(* PLC project Unnamed, Unknown Unnamed 1 *)
(* stored: creationDateTime 2026-03-27T23:35:05, modificationDateTime 2026-03-27T23:35:05 *)

PROGRAM main
  VAR
    start AT %IX0.0 : BOOL;
    stop AT %IX0.1 : BOOL;
    led AT %QX0.0 : BOOL;
  END_VAR
  VAR
    coil : BOOL;
    TON0 : TON;
    TOF0 : TOF;
  END_VAR

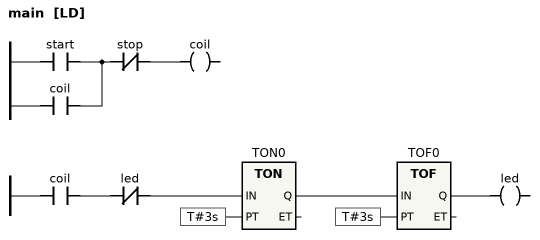
(* LD diagram, written out as Structured Text *)
coil := (start OR coil) AND NOT stop;
TON0(IN := coil AND NOT led, PT := T#3s);
TOF0(IN := TON0.Q, PT := T#3s);
led := TOF0.Q;
END_PROGRAM

CONFIGURATION Config0
  RESOURCE Res0 ON PLC
    TASK task0(INTERVAL := T#20ms, PRIORITY := 1);
    PROGRAM instance0 WITH task0 : main;
  END_RESOURCE
END_CONFIGURATION
